{attribute 'qualified_only'}
VAR_GLOBAL
	
(**************************************************** Granulowanie *****************************************************************)
	//*********************************************************************
	{attribute 'OPC.UA.DA' := '1'}
	{attribute 'OPC.UA.DA.StructuredType' := '1'}
	{attribute 'OPC.UA.DA.Description' := 'stGranHmi (structured) type '} 
	stGranHmi : ST_GranHmi;
	

	
END_VAR

(* stored: Version 1.1.0.1, ProductVersion 3.1.4024.15
   GVL GVL_Granulation: Id {25aebae5-868d-41b2-96cb-a96c8b42a7eb} *)
